FUNCTION_BLOCK TEST_MUL2 (* Test MUL functions *)
  (* Standard: IEC 61499-1 *)
  (* Version 0.0, 2006-09-11, JHC, Holobloc Inc *)
  (* Compiler header: package fb.rt.test; *)
  (* Compiler classdef: SimpleFB *)
  (* Compiler Java Sun JDK 1.5.0 *)
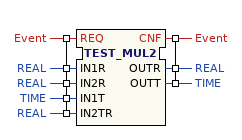
  EVENT_INPUT
    REQ WITH IN1R, IN2R, IN2TR, IN1T;
  END_EVENT
  EVENT_OUTPUT
    CNF WITH OUTR, OUTT;
  END_EVENT
  VAR_INPUT
    IN1R : REAL;
    IN2R : REAL;
    IN1T : TIME;
    IN2TR : REAL;
  END_VAR
  VAR_OUTPUT
    OUTR : REAL;
    OUTT : TIME;
  END_VAR
  ALGORITHM REQ IN FBD:
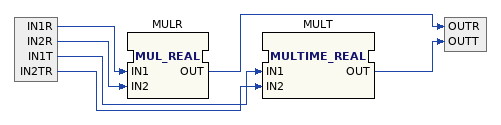
    FBS
      MULR : MUL_REAL;
      MULT : MULTIME_REAL;
    END_FBS
    DATA_CONNECTIONS
      IN1R TO MULR.IN1;
      IN2R TO MULR.IN2;
      MULR.OUT TO OUTR;
      IN1T TO MULT.IN1;
      MULT.OUT TO OUTT;
      IN2TR TO MULT.IN2;
    END_CONNECTIONS
  END_ALGORITHM
END_FUNCTION_BLOCK
